// LS Electric XG5000 project: 과년70_1_제안
// PLC NewPLC
// module base 0 slot 0: 입출력 모듈:XBC-DR20S (DC 24V 입력 12점, 릴레이 출력 8점)

PROGRAM NewProgram (task: 스캔 프로그램)

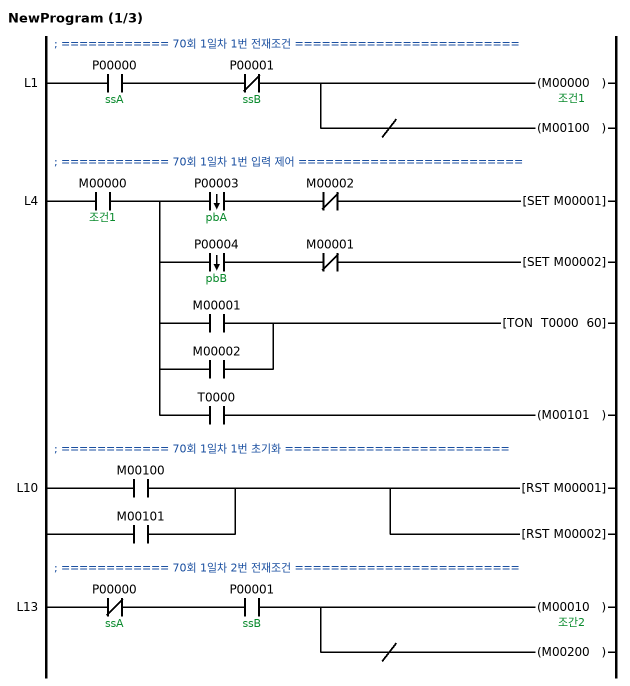
// ============ 70회 1일차 1번 전재조건 =========================
; L1
LOAD      P00000	// ssA
AND NOT   P00001	// ssB
OUT       M00000	// 조건1
NOT
OUT       M00100
// ============ 70회 1일차 1번 입력 제어 =========================
; L4
LOAD      M00000	// 조건1
MPUSH
ANDN      P00003	// pbA
AND NOT   M00002
SET       M00001
MLOAD
ANDN      P00004	// pbB
AND NOT   M00001
SET       M00002
MLOAD
LOAD      M00001
OR        M00002
AND LOAD
TON       T0000 60
MPOP
AND       T0000
OUT       M00101
// ============ 70회 1일차 1번 초기화 =========================
; L10
LOAD      M00100
OR        M00101
RST       M00001
RST       M00002
// ============ 70회 1일차 2번 전재조건 =========================
; L13
LOAD NOT  P00000	// ssA
AND       P00001	// ssB
OUT       M00010	// 조간2
NOT
OUT       M00200

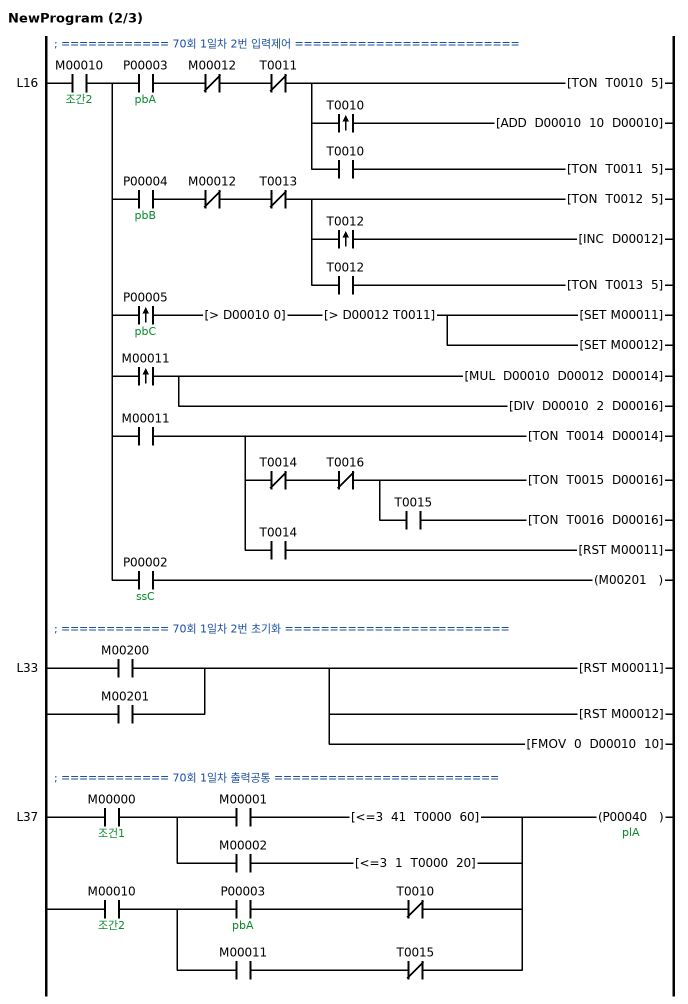
// ============ 70회 1일차 2번 입력제어 =========================
; L16
LOAD      M00010	// 조간2
MPUSH
AND       P00003	// pbA
AND NOT   M00012
AND NOT   T0011
TON       T0010 5
MPUSH
ANDP      T0010
ADD       D00010 10 D00010
MPOP
AND       T0010
TON       T0011 5
MLOAD
AND       P00004	// pbB
AND NOT   M00012
AND NOT   T0013
TON       T0012 5
MPUSH
ANDP      T0012
INC       D00012
MPOP
AND       T0012
TON       T0013 5
MLOAD
ANDP      P00005	// pbC
AND>      D00010 0
AND>      D00012 T0011
SET       M00011
SET       M00012
MLOAD
ANDP      M00011
MUL       D00010 D00012 D00014
DIV       D00010 2 D00016
MLOAD
AND       M00011
TON       T0014 D00014
MPUSH
AND NOT   T0014
AND NOT   T0016
TON       T0015 D00016
AND       T0015
TON       T0016 D00016
MPOP
AND       T0014
RST       M00011
MPOP
AND       P00002	// ssC
OUT       M00201
// ============ 70회 1일차 2번 초기화 =========================
; L33
LOAD      M00200
OR        M00201
RST       M00011
RST       M00012
FMOV      0 D00010 10
// ============ 70회 1일차 출력공통 =========================
; L37
LOAD      M00000	// 조건1
LOAD      M00001
AND<=3    41 T0000 60
LOAD      M00002
AND<=3    1 T0000 20
OR LOAD
AND LOAD
LOAD      M00010	// 조간2
LOAD      P00003	// pbA
AND NOT   T0010
LOAD      M00011
AND NOT   T0015
OR LOAD
AND LOAD
OR LOAD
OUT       P00040	// plA

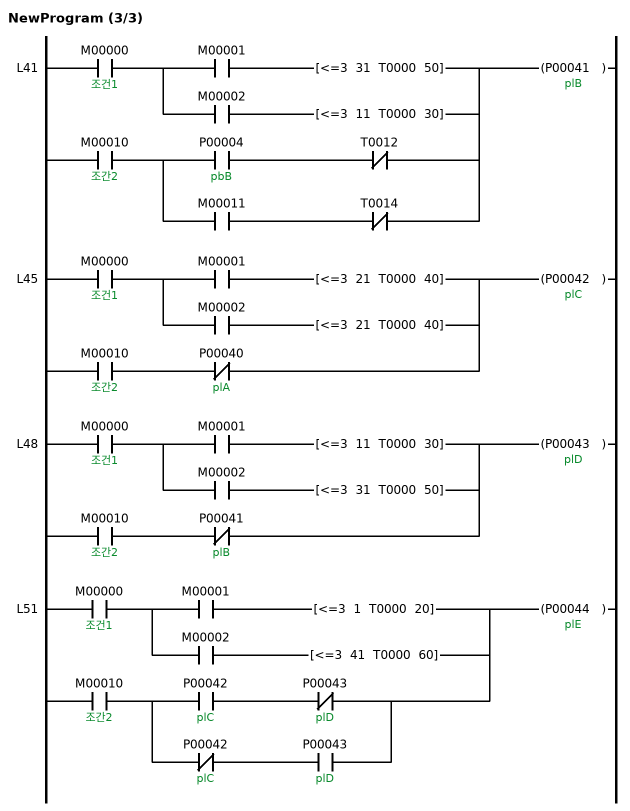
; L41
LOAD      M00000	// 조건1
LOAD      M00001
AND<=3    31 T0000 50
LOAD      M00002
AND<=3    11 T0000 30
OR LOAD
AND LOAD
LOAD      M00010	// 조간2
LOAD      P00004	// pbB
AND NOT   T0012
LOAD      M00011
AND NOT   T0014
OR LOAD
AND LOAD
OR LOAD
OUT       P00041	// plB
; L45
LOAD      M00000	// 조건1
LOAD      M00001
AND<=3    21 T0000 40
LOAD      M00002
AND<=3    21 T0000 40
OR LOAD
AND LOAD
LOAD      M00010	// 조간2
AND NOT   P00040	// plA
OR LOAD
OUT       P00042	// plC
; L48
LOAD      M00000	// 조건1
LOAD      M00001
AND<=3    11 T0000 30
LOAD      M00002
AND<=3    31 T0000 50
OR LOAD
AND LOAD
LOAD      M00010	// 조간2
AND NOT   P00041	// plB
OR LOAD
OUT       P00043	// plD
; L51
LOAD      M00000	// 조건1
LOAD      M00001
AND<=3    1 T0000 20
LOAD      M00002
AND<=3    41 T0000 60
OR LOAD
AND LOAD
LOAD      M00010	// 조간2
LOAD      P00042	// plC
AND NOT   P00043	// plD
LOAD NOT  P00042	// plC
AND       P00043	// plD
OR LOAD
AND LOAD
OR LOAD
OUT       P00044	// plE